FUNCTION_BLOCK Demux
  (* Version 1.0, 2007-08-28, Goran Cengic, Chalmers *)
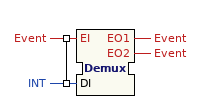
  EVENT_INPUT
    EI WITH DI;
  END_EVENT
  EVENT_OUTPUT
    EO1;
    EO2;
  END_EVENT
  VAR_INPUT
    DI : INT;
  END_VAR
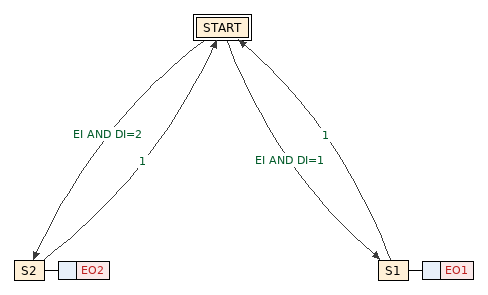
  EC_STATES
    START;
    S1 : -> EO1;
    S2 : -> EO2;
  END_STATES
  EC_TRANSITIONS
    START TO S1 := EI AND DI=1;
    S1 TO START := 1;
    START TO S2 := EI AND DI=2;
    S2 TO START := 1;
  END_TRANSITIONS
END_FUNCTION_BLOCK
